// TIA Portal V18 export
// export: Created 2026-06-08T16:32:20.5407716Z, ExportSetting WithDefaults, DisplayName Totally Integrated Automation Portal, DisplayVersion V18, DisplayName TIA Portal Openness, DisplayVersion V18, DisplayName TIA Portal Version Control Interface, DisplayVersion V18, DisplayName STEP 7 Professional, DisplayVersion V18, DisplayName STEP 7 Safety, DisplayVersion V18, DisplayName WinCC Professional, DisplayVersion V18
FUNCTION_BLOCK "LID_SORTING_STATION"   // FB3, LAD
VERSION : 0.1
// stored: AutoNumber true, IsIECCheckEnabled false, UDAEnableTagReadback false
BEGIN

REGION Network 1: BEGIN SORTING CONVYER
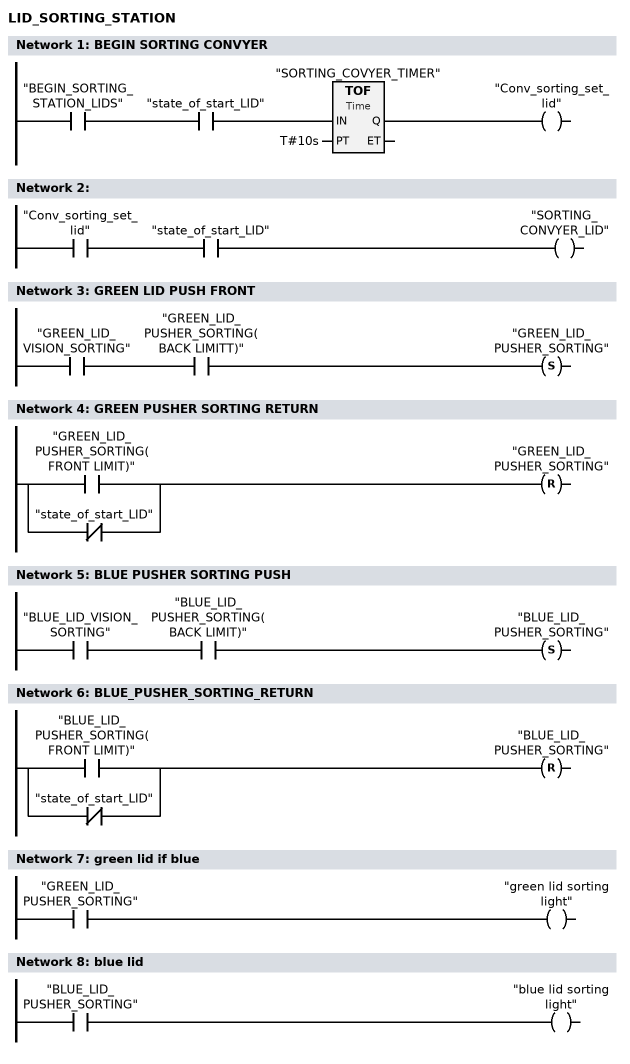
   RUNG wire#powerrail
      Contact( "BEGIN_SORTING_STATION_LIDS" )
      Contact( "state_of_start_LID" )
      { S7_Templates := "time_type := Time" } "SORTING_COVYER_TIMER".TOF(pt := T#10s, et =>)
      Coil( "Conv_sorting_set_lid" )
   END_RUNG
   // the same network as SCL:
   "SORTING_COVYER_TIMER".TOF(IN := "BEGIN_SORTING_STATION_LIDS" AND "state_of_start_LID", PT := T#10s);
   "Conv_sorting_set_lid" := "SORTING_COVYER_TIMER".Q;
END_REGION

REGION Network 2
   RUNG wire#powerrail
      Contact( "Conv_sorting_set_lid" )
      Contact( "state_of_start_LID" )
      Coil( "SORTING_CONVYER_LID" )
   END_RUNG
   // the same network as SCL:
   "SORTING_CONVYER_LID" := "Conv_sorting_set_lid" AND "state_of_start_LID";
END_REGION

REGION Network 3: GREEN LID PUSH FRONT
   RUNG wire#powerrail
      Contact( "GREEN_LID_VISION_SORTING" )
      Contact( "GREEN_LID_PUSHER_SORTING(BACK LIMITT)" )
      S_Coil( "GREEN_LID_PUSHER_SORTING" )
   END_RUNG
   // the same network as SCL:
   IF "GREEN_LID_VISION_SORTING" AND "GREEN_LID_PUSHER_SORTING(BACK LIMITT)" THEN
       "GREEN_LID_PUSHER_SORTING" := TRUE;
   END_IF;
END_REGION

REGION Network 4: GREEN PUSHER SORTING RETURN
   RUNG wire#powerrail
      Contact( "GREEN_LID_PUSHER_SORTING(FRONT LIMIT)" )
      wire#w1
      R_Coil( "GREEN_LID_PUSHER_SORTING" )
   END_RUNG
   RUNG wire#powerrail
      I_Contact( "state_of_start_LID" )
   END_RUNG wire#w1
   // the same network as SCL:
   IF "GREEN_LID_PUSHER_SORTING(FRONT LIMIT)" OR NOT "state_of_start_LID" THEN
       "GREEN_LID_PUSHER_SORTING" := FALSE;
   END_IF;
END_REGION

REGION Network 5: BLUE PUSHER SORTING PUSH
   RUNG wire#powerrail
      Contact( "BLUE_LID_VISION_SORTING" )
      Contact( "BLUE_LID_PUSHER_SORTING(BACK LIMIT)" )
      S_Coil( "BLUE_LID_PUSHER_SORTING" )
   END_RUNG
   // the same network as SCL:
   IF "BLUE_LID_VISION_SORTING" AND "BLUE_LID_PUSHER_SORTING(BACK LIMIT)" THEN
       "BLUE_LID_PUSHER_SORTING" := TRUE;
   END_IF;
END_REGION

REGION Network 6: BLUE_PUSHER_SORTING_RETURN
   RUNG wire#powerrail
      Contact( "BLUE_LID_PUSHER_SORTING(FRONT LIMIT)" )
      wire#w1
      R_Coil( "BLUE_LID_PUSHER_SORTING" )
   END_RUNG
   RUNG wire#powerrail
      I_Contact( "state_of_start_LID" )
   END_RUNG wire#w1
   // the same network as SCL:
   IF "BLUE_LID_PUSHER_SORTING(FRONT LIMIT)" OR NOT "state_of_start_LID" THEN
       "BLUE_LID_PUSHER_SORTING" := FALSE;
   END_IF;
END_REGION

REGION Network 7: green lid if blue
   RUNG wire#powerrail
      Contact( "GREEN_LID_PUSHER_SORTING" )
      Coil( "green lid sorting light" )
   END_RUNG
   // the same network as SCL:
   "green lid sorting light" := "GREEN_LID_PUSHER_SORTING";
END_REGION

REGION Network 8: blue lid
   RUNG wire#powerrail
      Contact( "BLUE_LID_PUSHER_SORTING" )
      Coil( "blue lid sorting light" )
   END_RUNG
   // the same network as SCL:
   "blue lid sorting light" := "BLUE_LID_PUSHER_SORTING";
END_REGION
END_FUNCTION_BLOCK
